FUNCTION_BLOCK TaskBaseExtended EXTENDS TaskBase
VAR_INPUT
END_VAR
VAR_OUTPUT
END_VAR
VAR
END_VAR

END_FUNCTION_BLOCK

(* stored: Version 1.1.0.1
   POU TaskBaseExtended: Id {e0c056f8-c6cc-066f-2ca2-1bd2036ca95d}, SpecialFunc None *)
